{attribute 'GeneratedUsingTerminal: AX8118-0100-0101-0101'}
{attribute addProperty BoxType "AX8118-0100-0101-0101"}
{attribute addProperty Id "DeviceDevice_6E2575772Device_SafetyDevice_Safety_C21945A160Ch_ACh_A_1FF86D8522WcStateAT %I*WcState_B516A2644InfoDataAT %I*InfoData_358A59CF25"}
{attribute addProperty CRC "2190976545"}
{attribute addProperty Size "113"}
TYPE AX8118_8297A621 :
STRUCT
	{attribute addProperty Name "Device"}
	Device : Device_6E257577;
	{attribute addProperty Name "Device_Safety"}
	Device_Safety : Device_Safety_C21945A1;
	{attribute addProperty Name "Ch_A"}
	Ch_A : Ch_A_1FF86D85;
	{attribute addProperty Name "WcState"}
	WcState : WcState_B516A264;
	{attribute addProperty Name "InfoData"}
	InfoData : InfoData_358A59CF;
END_STRUCT
END_TYPE

(* stored: Version 1.2.0.0, ProductVersion 3.1.4024.9
   DUT AX8118_8297A621: Id {3b970dbd-654a-407b-b5a7-842d5cd5cfb3} *)
